INTERFACE I_NodePack

METHOD PUBLIC RegisterWithGraph
VAR_INPUT
	TcGraph : I_GraphFactory;
END_VAR
END_METHOD

END_INTERFACE

(* stored: Version 1.1.0.1, ProductVersion 3.1.4024.12
   Itf I_NodePack: Id {30b9a38a-1df6-0049-1a2e-20ebc2a31c34}
   Method RegisterWithGraph: Id {08c57c3e-0a8f-06be-0ca2-d87069d7f01b} *)
